// TIA Portal V15.1 export
// export: Created 2024-06-21T08:41:05.3670031Z, ExportSetting WithDefaults, DisplayName Totally Integrated Automation Portal, DisplayVersion V15.1 Update 5, DisplayName TIA Portal Openness, DisplayVersion V15.1 Update 5, DisplayName SINAMICS Startdrive Advanced, DisplayVersion V15.1, DisplayName G130, G150, S120, S150, SINAMICS MV, S210, DisplayVersion V15.1, DisplayName G110M, G120, G120C, G120D, G120P, DisplayVersion V15.1, DisplayName STEP 7 Professional, DisplayVersion V15.1 Update 5, DisplayName STEP 7 Safety, DisplayVersion V15.1, DisplayName WinCC Professional, DisplayVersion V15.1 Update 5, DisplayName SIMATIC Visualization Architect, DisplayVersion V15.1
FUNCTION_BLOCK "LProcPAC"   // FB1740, FBD
TITLE = LProcPAC
{ S7_Optimized_Access := 'TRUE' }
AUTHOR : CSTAAL
VERSION : 0.1
// This module handles the power measuring device
// stored: AutoNumber false, IsIECCheckEnabled false, IsRetainMemResEnabled false, MemoryReserve 100, SetENOAutomatically False, UDAEnableTagReadback false
   VAR_INPUT
      I_HWSubModule { ExternalAccessible := 'False'; ExternalVisible := 'False'; ExternalWritable := 'False'} : HW_SUBMODULE;   // Connection with Hardware Sub Module
   END_VAR
   VAR_OUTPUT
      O_ControlBytes { ExternalAccessible := 'False'; ExternalVisible := 'False'; ExternalWritable := 'False'} : Word;   // Control Bytes for the PAC
      O_AlarmA { ExternalAccessible := 'False'; ExternalVisible := 'False'; ExternalWritable := 'False'} : Bool;   // Alarm A
      O_AlarmB { ExternalAccessible := 'False'; ExternalVisible := 'False'; ExternalWritable := 'False'} : Bool;   // Alarm B
      O_AlarmC { ExternalAccessible := 'False'; ExternalVisible := 'False'; ExternalWritable := 'False'} : Bool;   // Alarm C
      O_AlarmD { ExternalAccessible := 'False'; ExternalVisible := 'False'; ExternalWritable := 'False'} : Bool;   // Alarm D
      O_AlarmABCondition { ExternalAccessible := 'False'; ExternalVisible := 'False'; ExternalWritable := 'False'} : Bool;   // Alarms resetable
      H_IAnim { ExternalAccessible := 'False'; ExternalVisible := 'False'; ExternalWritable := 'False'} : Word;   // Animation bits to Icon in WinCC
      H_AlarmWord { ExternalAccessible := 'False'; ExternalVisible := 'False'; ExternalWritable := 'False'} : DWord;   // Alarm Word
   END_VAR
   VAR DB_SPECIFIC
      Cmd { ExternalAccessible := 'False'; ExternalVisible := 'False'; ExternalWritable := 'False'} : Struct   // Command (copied from HMI Command) / Command
         Reset_min_max_Data { ExternalAccessible := 'False'; ExternalVisible := 'False'; ExternalWritable := 'False'} : Bool := FALSE;   // 0 / Reset_min_max_Data
         Reset_Energy_Meter { ExternalAccessible := 'False'; ExternalVisible := 'False'; ExternalWritable := 'False'} : Bool := FALSE;   // 1 / Reset_Energy_Meter
      END_STRUCT;
   END_VAR
   VAR
      C_UnitAmps { ExternalAccessible := 'False'; ExternalVisible := 'False'; ExternalWritable := 'False'} : Int;   // Unit Amps (1 = mA; 2 = kA)
      C_UnitVolts { ExternalAccessible := 'False'; ExternalVisible := 'False'; ExternalWritable := 'False'} : Int;   // Unit Volts (1 = mV; 2 = V)
      C_UnitWatts { ExternalAccessible := 'False'; ExternalVisible := 'False'; ExternalWritable := 'False'} : Int;   // Unit Watts (1 = W; 2 = kW)
      Units { ExternalAccessible := 'False'; ExternalVisible := 'False'; ExternalWritable := 'False'} : Struct   // Units
         "Amps-mA" { ExternalAccessible := 'False'; ExternalVisible := 'False'; ExternalWritable := 'False'} : Bool;   // Amps in mA
         "Amps-kA" { ExternalAccessible := 'False'; ExternalVisible := 'False'; ExternalWritable := 'False'} : Bool;   // Amps in kA
         "Volts-mV" { ExternalAccessible := 'False'; ExternalVisible := 'False'; ExternalWritable := 'False'} : Bool;   // Volts in mV
         "Volts-kV" { ExternalAccessible := 'False'; ExternalVisible := 'False'; ExternalWritable := 'False'} : Bool;   // Volts in kV
         "Watts-W" { ExternalAccessible := 'False'; ExternalVisible := 'False'; ExternalWritable := 'False'} : Bool;   // Watts in W
         "Watts-kW" { ExternalAccessible := 'False'; ExternalVisible := 'False'; ExternalWritable := 'False'} : Bool;   // Watts in kW
      END_STRUCT;
      H_HMICmd : Word;   // HMI Command
   END_VAR
   VAR DB_SPECIFIC
      H_Out : Struct   // HMI
         Anim : Word;   // HMI Animation of the object
         DBnr : Int;   // HMI Animation DB number
         U12 : Real;   // Voltage L1-L2
         U23 : Real;   // Voltage L2-L3
         U31 : Real;   // Voltage L3-L1
         U12Max : Real;   // MAX Voltage L1-L2
         U23Max : Real;   // MAX Voltage L2-L3
         U31Max : Real;   // MAX Voltage L3-L1
         UL1 : Real;   // UL1
         UL2 : Real;   // UL2
         UL3 : Real;   // UL3
         UL1Max : Real;   // MAX Voltage L1
         UL2Max : Real;   // MAX Voltage L2
         UL3Max : Real;   // MAX Voltage L3
         I1 : Real;   // Current L1
         I2 : Real;   // Current L2
         I3 : Real;   // Current L3
         I1Max : Real;   // MAX Current L1
         I2Max : Real;   // MAX Current L2
         I3Max : Real;   // MAX Current L3
         PTotal : Real;   // Total active power
         PTotalMax : Real;   // Total MAX active power
      END_STRUCT;
   END_VAR
   VAR
      AlarmA { ExternalAccessible := 'False'; ExternalVisible := 'False'; ExternalWritable := 'False'} : Bool;   // Alarm A
      AlarmB { ExternalAccessible := 'False'; ExternalVisible := 'False'; ExternalWritable := 'False'} : Bool;   // Alarm B
      AlarmC { ExternalAccessible := 'False'; ExternalVisible := 'False'; ExternalWritable := 'False'} : Bool;   // Alarm C
      AlarmD { ExternalAccessible := 'False'; ExternalVisible := 'False'; ExternalWritable := 'False'} : Bool;   // Alarm D
      AlarmABCondition { ExternalAccessible := 'False'; ExternalVisible := 'False'; ExternalWritable := 'False'} : Bool;   // Alarm AB condition
   END_VAR
   VAR DB_SPECIFIC
      DBnr { ExternalAccessible := 'False'; ExternalVisible := 'False'; ExternalWritable := 'False'} : Int;   // HMI DB number
   END_VAR
   VAR
      _PACDriver { ExternalAccessible := 'False'; ExternalVisible := 'False'; ExternalWritable := 'False'} : "LProcPAC-Driver";   // FB
      _PACVisu { ExternalAccessible := 'False'; ExternalVisible := 'False'; ExternalWritable := 'False'} : "LProcPAC-Visu";   // FB
   END_VAR
   VAR_TEMP
      ControlBytes : Word;   // Control Bytes for the PAC
      L12 : Real;   // Temporary test variable
      L23 : Real;   // Temporary test variable
      L31 : Real;   // Temporary test variable
   END_VAR
   VAR_TEMP   // added for the SCL form of the ladder/FBD networks
      _w1 : Bool;
   END_VAR
BEGIN

NETWORK
TITLE = **** 1 - Inputs **** DB number
// DB number
      L     DINO;
      T     #DBnr;

REGION Network 2: **** 1 - Inputs **** HMI Commands
   // HMI Commands
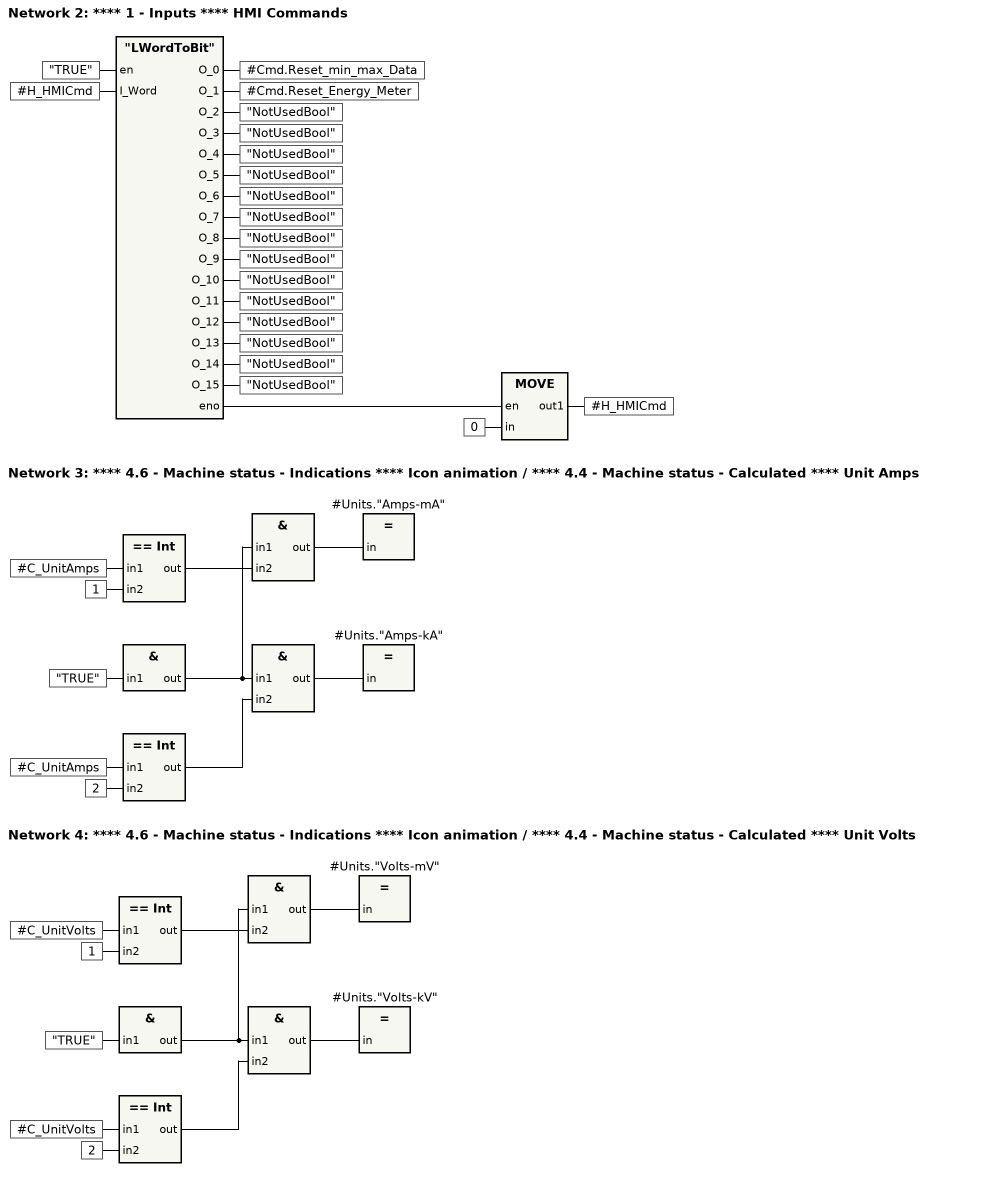
   "LWordToBit"(EN := "TRUE",
                I_Word := #H_HMICmd,
                O_0 => #Cmd.Reset_min_max_Data,
                O_1 => #Cmd.Reset_Energy_Meter,
                O_2 => "NotUsedBool",
                O_3 => "NotUsedBool",
                O_4 => "NotUsedBool",
                O_5 => "NotUsedBool",
                O_6 => "NotUsedBool",
                O_7 => "NotUsedBool",
                O_8 => "NotUsedBool",
                O_9 => "NotUsedBool",
                O_10 => "NotUsedBool",
                O_11 => "NotUsedBool",
                O_12 => "NotUsedBool",
                O_13 => "NotUsedBool",
                O_14 => "NotUsedBool",
                O_15 => "NotUsedBool",
                ENO => #_w1);
   IF #_w1 THEN #H_HMICmd := 0; END_IF;
END_REGION

REGION Network 3: **** 4.6 - Machine status - Indications **** Icon animation / **** 4.4 - Machine status - Calculated **** Unit Amps
   // Icon animation to WinCC / Unit Amps
   #Units."Amps-mA" := "TRUE" AND (#C_UnitAmps = 1);
   #Units."Amps-kA" := "TRUE" AND (#C_UnitAmps = 2);
END_REGION

REGION Network 4: **** 4.6 - Machine status - Indications **** Icon animation / **** 4.4 - Machine status - Calculated **** Unit Volts
   // Icon animation to WinCC / Unit Volts
   #Units."Volts-mV" := "TRUE" AND (#C_UnitVolts = 1);
   #Units."Volts-kV" := "TRUE" AND (#C_UnitVolts = 2);
END_REGION

REGION Network 5: **** 4.6 - Machine status - Indications **** Icon animation / **** 4.4 - Machine status - Calculated **** Unit Watts
   // Icon animation to WinCC / Unit Watts
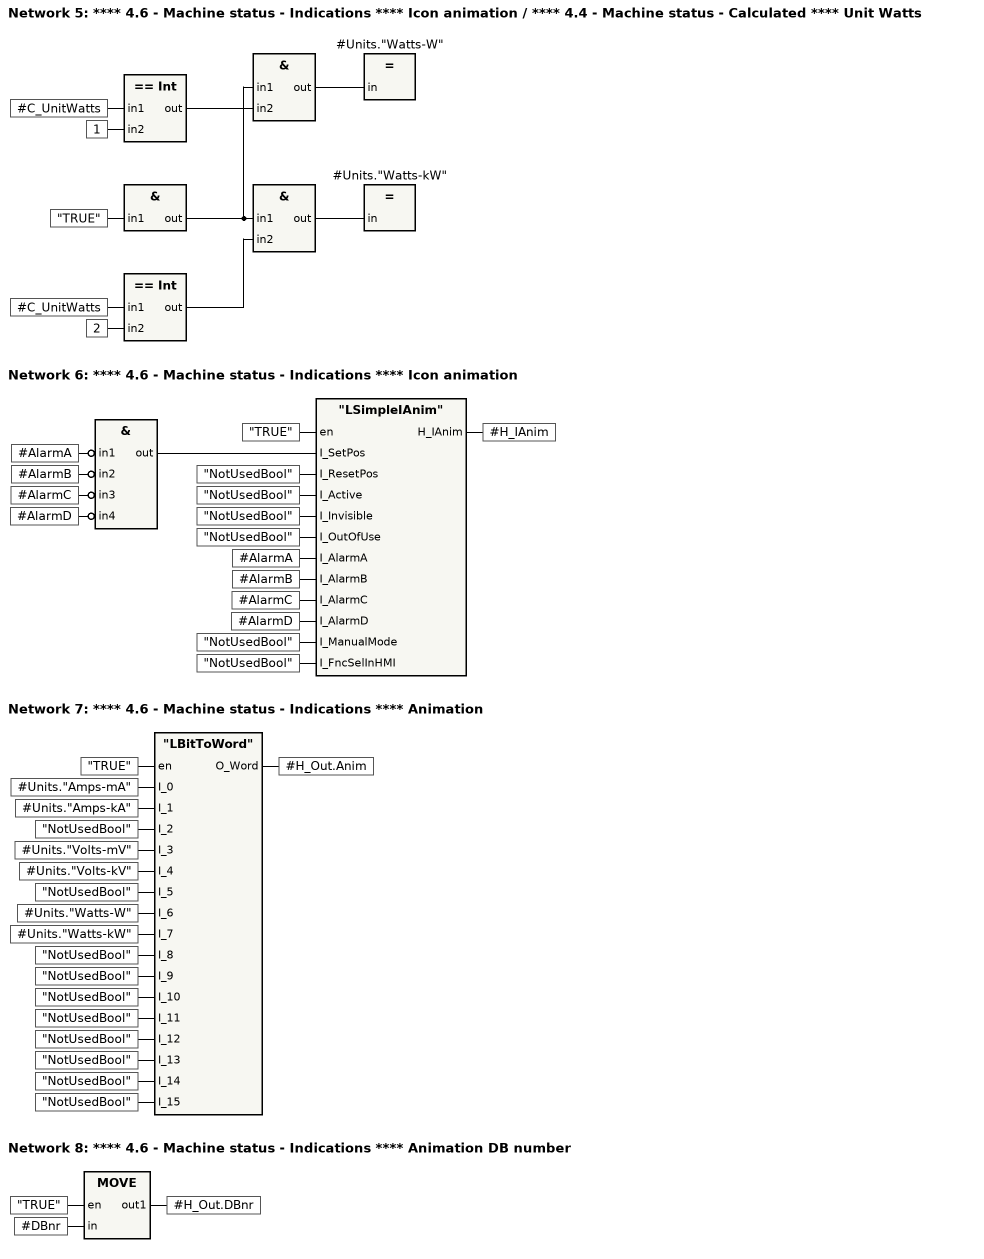
   #Units."Watts-W" := "TRUE" AND (#C_UnitWatts = 1);
   #Units."Watts-kW" := "TRUE" AND (#C_UnitWatts = 2);
END_REGION

REGION Network 6: **** 4.6 - Machine status - Indications **** Icon animation
   // Icon animation to WinCC / Icon animation
   IF "TRUE" THEN
       "LSimpleIAnim"(I_SetPos := NOT #AlarmA AND NOT #AlarmB AND NOT #AlarmC AND NOT #AlarmD,
                      I_ResetPos := "NotUsedBool",
                      I_Active := "NotUsedBool",
                      I_Invisible := "NotUsedBool",
                      I_OutOfUse := "NotUsedBool",
                      I_AlarmA := #AlarmA,
                      I_AlarmB := #AlarmB,
                      I_AlarmC := #AlarmC,
                      I_AlarmD := #AlarmD,
                      I_ManualMode := "NotUsedBool",
                      I_FncSelInHMI := "NotUsedBool",
                      H_IAnim => #H_IAnim);
   END_IF;
END_REGION

REGION Network 7: **** 4.6 - Machine status - Indications **** Animation
   // Animation
   IF "TRUE" THEN
       "LBitToWord"(I_0 := #Units."Amps-mA",
                    I_1 := #Units."Amps-kA",
                    I_2 := "NotUsedBool",
                    I_3 := #Units."Volts-mV",
                    I_4 := #Units."Volts-kV",
                    I_5 := "NotUsedBool",
                    I_6 := #Units."Watts-W",
                    I_7 := #Units."Watts-kW",
                    I_8 := "NotUsedBool",
                    I_9 := "NotUsedBool",
                    I_10 := "NotUsedBool",
                    I_11 := "NotUsedBool",
                    I_12 := "NotUsedBool",
                    I_13 := "NotUsedBool",
                    I_14 := "NotUsedBool",
                    I_15 := "NotUsedBool",
                    O_Word => #H_Out.Anim);
   END_IF;
END_REGION

REGION Network 8: **** 4.6 - Machine status - Indications **** Animation DB number
   // Animation DB number
   IF "TRUE" THEN #H_Out.DBnr := #DBnr; END_IF;
END_REGION

REGION Network 9: **** 7.1 SubModules - Non Machine **** Method 2: PAC3200 Driver
   // PAC3200 Driver
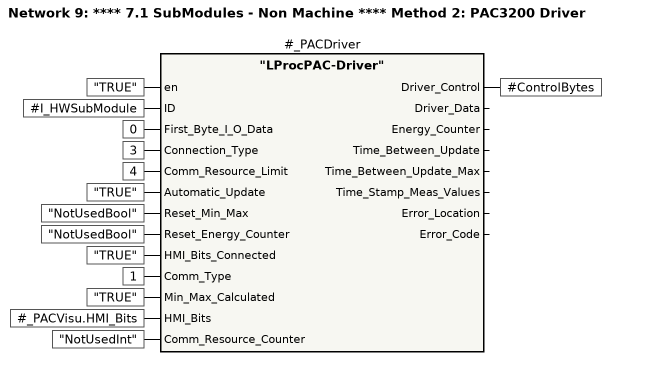
   IF "TRUE" THEN
       #_PACDriver(ID := #I_HWSubModule,   // "LProcPAC-Driver"
                   First_Byte_I_O_Data := 0,
                   Connection_Type := 3,
                   Comm_Resource_Limit := 4,
                   Automatic_Update := "TRUE",
                   Reset_Min_Max := "NotUsedBool",
                   Reset_Energy_Counter := "NotUsedBool",
                   HMI_Bits_Connected := "TRUE",
                   Comm_Type := 1,
                   Min_Max_Calculated := "TRUE",
                   HMI_Bits := #_PACVisu.HMI_Bits,
                   Comm_Resource_Counter := "NotUsedInt",
                   Driver_Control => #ControlBytes);
   END_IF;
END_REGION

REGION Network 10: **** 7.1 SubModules - Non Machine **** Method 2: PAC3200 Visualisation
   // PAC3200 Visualisation
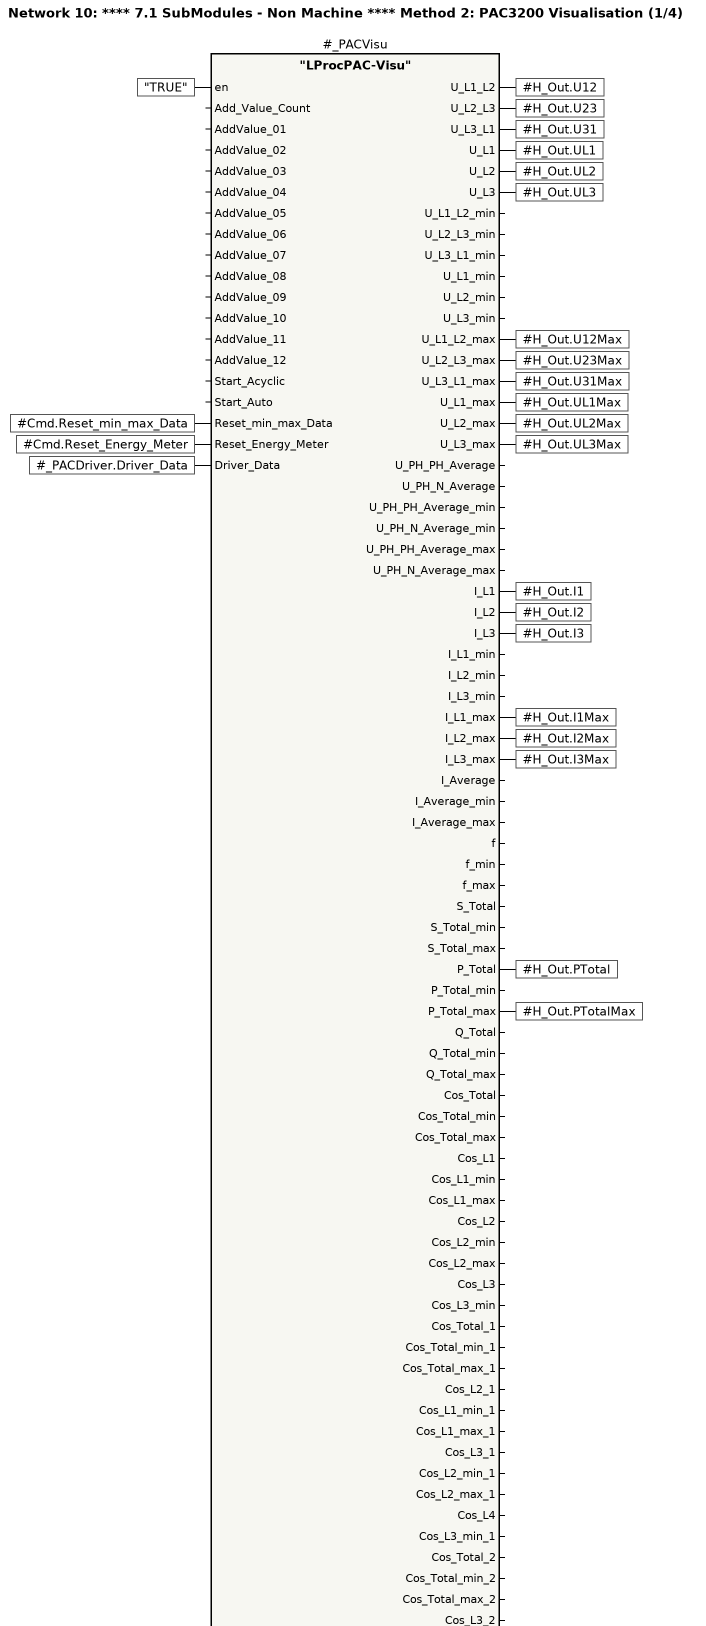
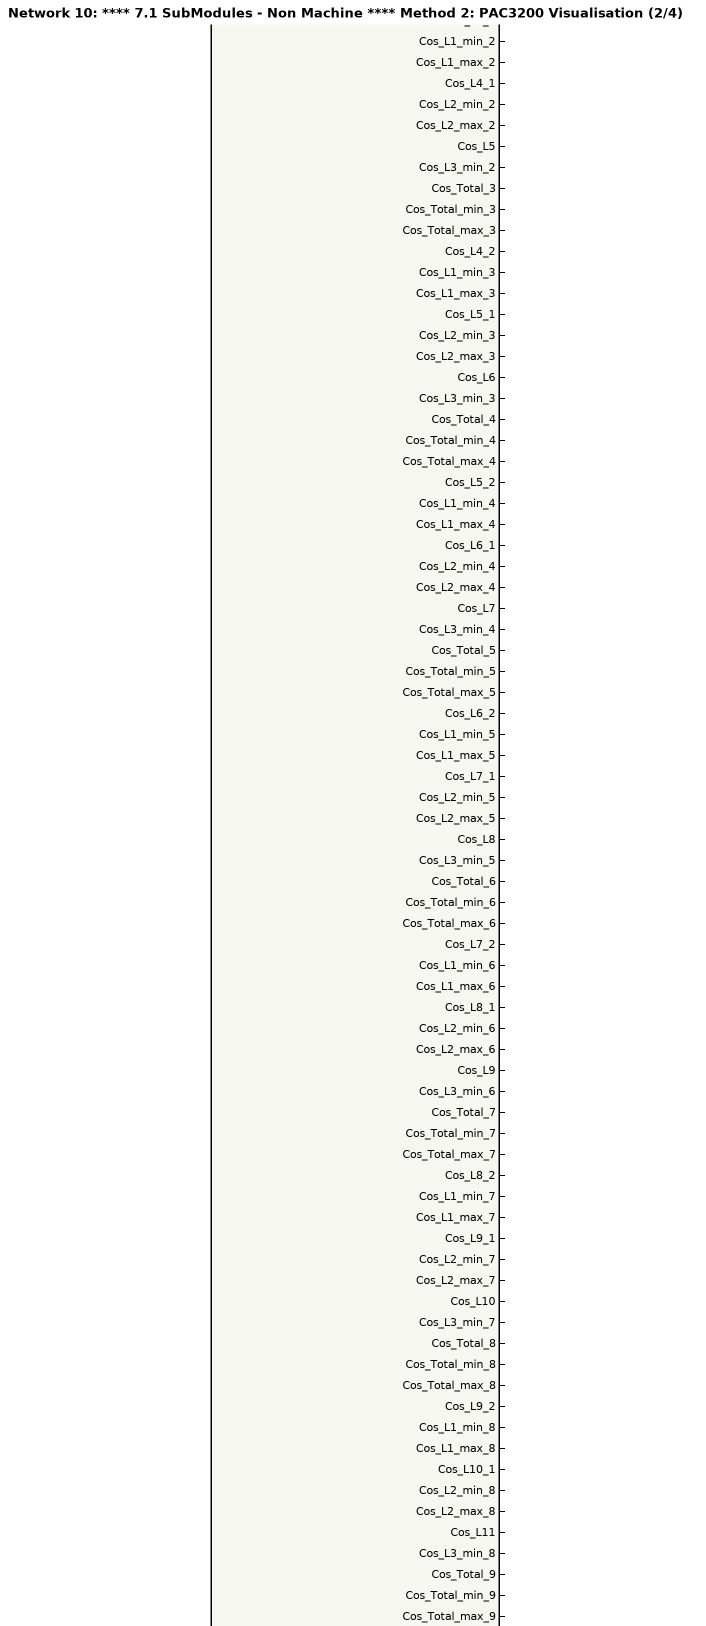
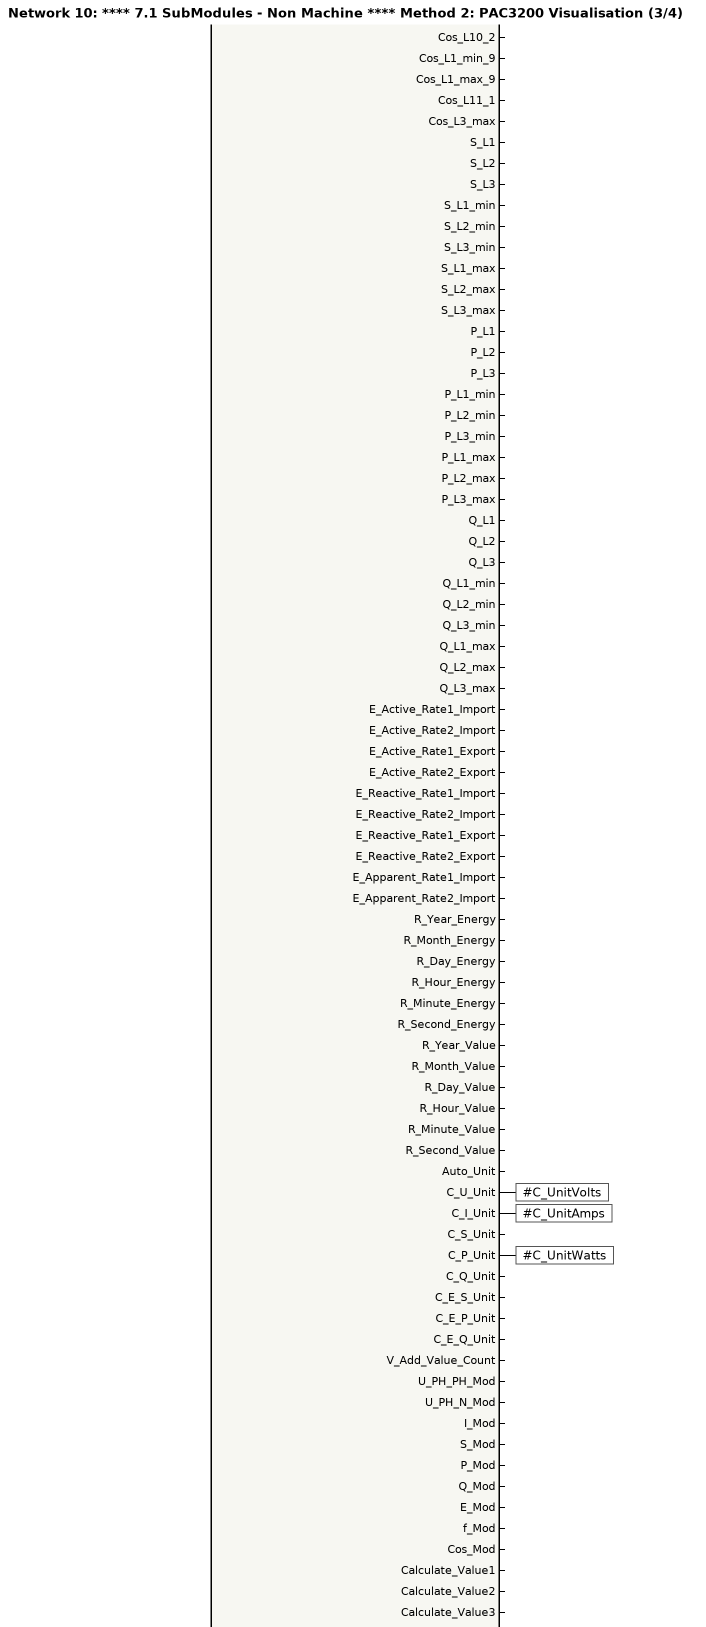
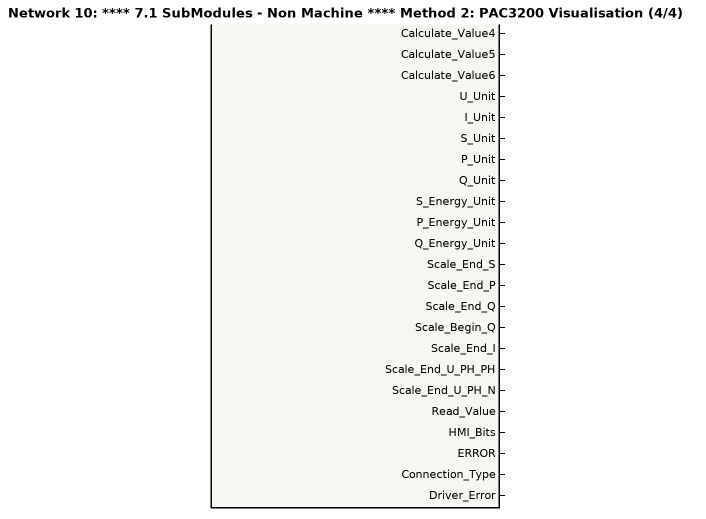
   IF "TRUE" THEN
       #_PACVisu(Reset_min_max_Data := #Cmd.Reset_min_max_Data,   // "LProcPAC-Visu"
                 Reset_Energy_Meter := #Cmd.Reset_Energy_Meter,
                 Driver_Data := #_PACDriver.Driver_Data,
                 U_L1_L2 => #H_Out.U12,
                 U_L2_L3 => #H_Out.U23,
                 U_L3_L1 => #H_Out.U31,
                 U_L1 => #H_Out.UL1,
                 U_L2 => #H_Out.UL2,
                 U_L3 => #H_Out.UL3,
                 U_L1_L2_max => #H_Out.U12Max,
                 U_L2_L3_max => #H_Out.U23Max,
                 U_L3_L1_max => #H_Out.U31Max,
                 U_L1_max => #H_Out.UL1Max,
                 U_L2_max => #H_Out.UL2Max,
                 U_L3_max => #H_Out.UL3Max,
                 I_L1 => #H_Out.I1,
                 I_L2 => #H_Out.I2,
                 I_L3 => #H_Out.I3,
                 I_L1_max => #H_Out.I1Max,
                 I_L2_max => #H_Out.I2Max,
                 I_L3_max => #H_Out.I3Max,
                 P_Total => #H_Out.PTotal,
                 P_Total_max => #H_Out.PTotalMax,
                 C_U_Unit => #C_UnitVolts,
                 C_I_Unit => #C_UnitAmps,
                 C_P_Unit => #C_UnitWatts);
   END_IF;
END_REGION

REGION Network 11: *** 8 - Outputs **** Control Bytes PAC
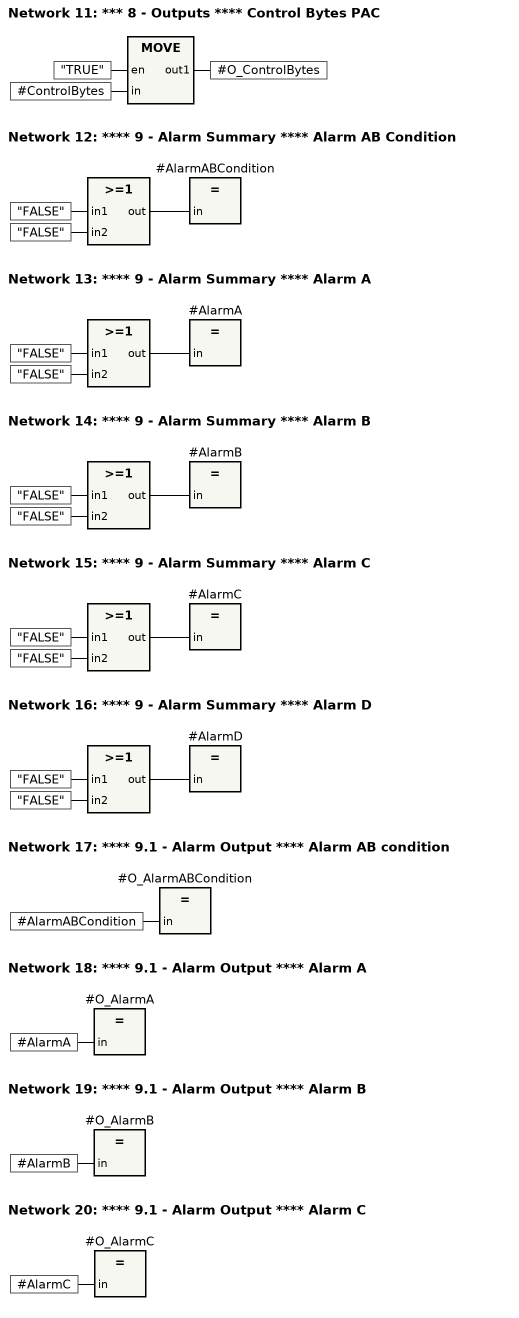
   IF "TRUE" THEN #O_ControlBytes := #ControlBytes; END_IF;
END_REGION

REGION Network 12: **** 9 - Alarm Summary **** Alarm AB Condition
   #AlarmABCondition := "FALSE" OR "FALSE";
END_REGION

REGION Network 13: **** 9 - Alarm Summary **** Alarm A
   #AlarmA := "FALSE" OR "FALSE";
END_REGION

REGION Network 14: **** 9 - Alarm Summary **** Alarm B
   #AlarmB := "FALSE" OR "FALSE";
END_REGION

REGION Network 15: **** 9 - Alarm Summary **** Alarm C
   #AlarmC := "FALSE" OR "FALSE";
END_REGION

REGION Network 16: **** 9 - Alarm Summary **** Alarm D
   #AlarmD := "FALSE" OR "FALSE";
END_REGION

REGION Network 17: **** 9.1 - Alarm Output **** Alarm AB condition
   // Alarm AB condition
   #O_AlarmABCondition := #AlarmABCondition;
END_REGION

REGION Network 18: **** 9.1 - Alarm Output **** Alarm A
   // Output Alarm A
   #O_AlarmA := #AlarmA;
END_REGION

REGION Network 19: **** 9.1 - Alarm Output **** Alarm B
   // Output Alarm B
   #O_AlarmB := #AlarmB;
END_REGION

REGION Network 20: **** 9.1 - Alarm Output **** Alarm C
   // Output Alarm A
   #O_AlarmC := #AlarmC;
END_REGION

REGION Network 21: **** 9.1 - Alarm Output **** Alarm D
   // Output Alarm D
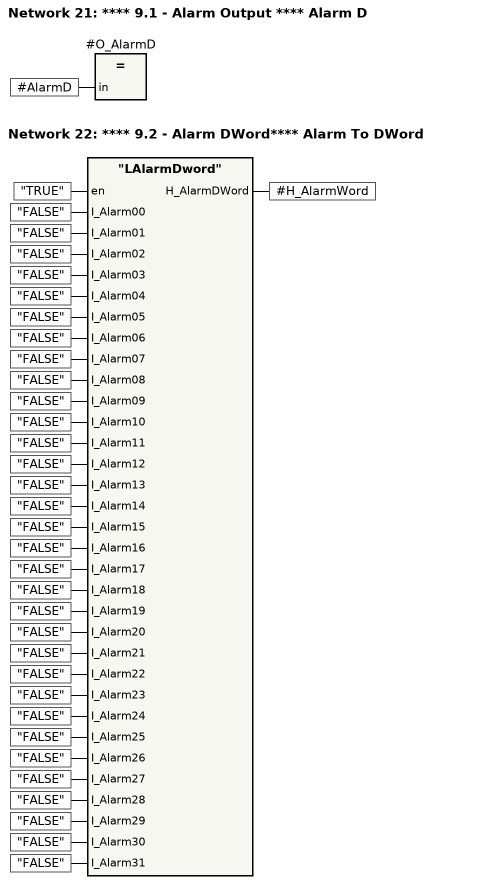
   #O_AlarmD := #AlarmD;
END_REGION

REGION Network 22: **** 9.2 - Alarm DWord**** Alarm To DWord
   // Alarm Word
   IF "TRUE" THEN
       "LAlarmDword"(I_Alarm00 := "FALSE",
                     I_Alarm01 := "FALSE",
                     I_Alarm02 := "FALSE",
                     I_Alarm03 := "FALSE",
                     I_Alarm04 := "FALSE",
                     I_Alarm05 := "FALSE",
                     I_Alarm06 := "FALSE",
                     I_Alarm07 := "FALSE",
                     I_Alarm08 := "FALSE",
                     I_Alarm09 := "FALSE",
                     I_Alarm10 := "FALSE",
                     I_Alarm11 := "FALSE",
                     I_Alarm12 := "FALSE",
                     I_Alarm13 := "FALSE",
                     I_Alarm14 := "FALSE",
                     I_Alarm15 := "FALSE",
                     I_Alarm16 := "FALSE",
                     I_Alarm17 := "FALSE",
                     I_Alarm18 := "FALSE",
                     I_Alarm19 := "FALSE",
                     I_Alarm20 := "FALSE",
                     I_Alarm21 := "FALSE",
                     I_Alarm22 := "FALSE",
                     I_Alarm23 := "FALSE",
                     I_Alarm24 := "FALSE",
                     I_Alarm25 := "FALSE",
                     I_Alarm26 := "FALSE",
                     I_Alarm27 := "FALSE",
                     I_Alarm28 := "FALSE",
                     I_Alarm29 := "FALSE",
                     I_Alarm30 := "FALSE",
                     I_Alarm31 := "FALSE",
                     H_AlarmDWord => #H_AlarmWord);
   END_IF;
END_REGION
END_FUNCTION_BLOCK
